FUNCTION HLI3_GetVEChannelBooleanValue : BOOL
VAR_INPUT
	/// HLI Channel Index
	nChanIdx: INT;
	/// Index of variable  range 1 ...     HLI_VE_VALUEMAX 
	nVEIndex: DINT;
	/// Array index. 0 if no array 
	nArrayIndex: DINT := 0;
	/// serves acess to the global variable array 
	bGlobal: BOOL;
END_VAR
VAR
	pVeData: POINTER TO VEData := 0;
	/// Size of the datatype of the returned value 
	iDatatypeSize: DINT;
	ptr: POINTER TO BOOL;
	ChIdx: UDINT;
	SizeField: DINT := 0;
END_VAR

(* ========================================================= *)
(*    FUN: GetVEChannelDINTValue                            *)
(* --------------------------------------------------------- *)
(*   Desc: Reads a V.E.Variable of Boolean                   *)
(* 	 Author: CL  / TV                                        *)
(*   Date: 16.05.2006                                        *)
(*   Last: 05.12.2013                                        *)
(*   Rev.: 1.3                                               *)
(* ========================================================= *)

IF  nVEIndex >= 0 AND
	nArrayIndex >= 0 THEN

	(* test if channel specific or global *)
	IF bGlobal = FALSE  THEN
		IF NOT HLI3_CheckChannelValid(nChannel := nChanIdx) THEN
			RETURN;
		END_IF
				
		pVeData := gpVECh[nChanIdx];
	ELSE
		pVeData := gpVEGlobal;
	END_IF

	IF pVeData <> 0 THEN
		IF pVeData <> 0 THEN
			iDatatypeSize := SIZEOF(ptr^);
                         	ptr := pVeData +  24  * nVEIndex + (iDatatypeSize * nArrayIndex);
                           HLI3_GetVEChannelBooleanValue := ptr^; (* successfully completed return *)
                END_IF
	END_IF
END_IF

END_FUNCTION

(* stored: Version 1.1.0.1, ProductVersion 3.1.4018.2
   POU HLI3_GetVEChannelBooleanValue: Id {c8758ad7-c4a9-4d7a-81e6-248b9273a457}, SpecialFunc None *)
